PROGRAM MAIN
VAR
END_VAR

Prg_NonInstantFunc();

END_PROGRAM

(* stored: Version 1.1.0.1, ProductVersion 3.1.4024.9
   POU MAIN: Id {be76b349-05ea-4870-8ace-088ca1cfd0cb}, SpecialFunc None *)
